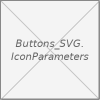
VISUALIZATION ButtonParameters  // 100x100
VAR_IN_OUT
	bState : BOOL;
END_VAR
    Frame (0,0 100x100)
        shows ButtonTemplate(bActive := bState)
    Image (0,0 100x100), image: Buttons_SVG.IconParameters
        OnMouseDown: execute { GVL_HMI.fbHMIControl.eScreenRequest := E_BaseVisu.Parameter; }
END_VISUALIZATION

(* stored: Version 1.1.0.1, ProductVersion 3.1.4024.11
   Visu ButtonParameters: Id {3e4e12fe-e12e-4f8e-9aa1-a489ae74e827} *)
